(* IEC 61131-3 sources: plc_generation_empirical_study/datasets/task_bank_c06_formal_core_runtime_v0_4/tasks/C06_W25_lean_composite, 2 files *)

(* ---- interface.st ---- *)
FUNCTION_BLOCK C06_W25_lean_composite
VAR_INPUT
    A_Ch1 : BOOL;
    A_Ch2 : BOOL;
    A_Ch3 : BOOL;
    A_AutoMode : BOOL;
    A_AutoRequest : BOOL;
    A_ManualRequest : BOOL;
    A_BypassRequest : BOOL;
    A_BypassPermit : BOOL;
    A_SafetyOK : BOOL;
    A_Reset : BOOL;
    B_ItemPulse : BOOL;
    B_Rejected : BOOL;
    B_Stop : BOOL;
    B_Reset : BOOL;
    B_Target : INT;
    B_RejectLimit : INT;
    SubsystemBEnable : BOOL;
    CrossReset : BOOL;
END_VAR
VAR_OUTPUT
    A_RunPermit : BOOL;
    A_Degraded : BOOL;
    A_BypassActive : BOOL;
    A_Blocked : BOOL;
    B_AcceptedCount : INT;
    B_RejectCount : INT;
    B_ConsecutiveRejects : INT;
    B_Complete : BOOL;
    B_LockedOut : BOOL;
    CrossReady : BOOL;
    CrossBlocked : BOOL;
END_VAR
END_FUNCTION_BLOCK

(* ---- reference.st ---- *)
FUNCTION_BLOCK C06_W25_lean_composite
VAR_INPUT
    A_Ch1 : BOOL;
    A_Ch2 : BOOL;
    A_Ch3 : BOOL;
    A_AutoMode : BOOL;
    A_AutoRequest : BOOL;
    A_ManualRequest : BOOL;
    A_BypassRequest : BOOL;
    A_BypassPermit : BOOL;
    A_SafetyOK : BOOL;
    A_Reset : BOOL;
    B_ItemPulse : BOOL;
    B_Rejected : BOOL;
    B_Stop : BOOL;
    B_Reset : BOOL;
    B_Target : INT;
    B_RejectLimit : INT;
    SubsystemBEnable : BOOL;
    CrossReset : BOOL;
END_VAR
VAR_OUTPUT
    A_RunPermit : BOOL;
    A_Degraded : BOOL;
    A_BypassActive : BOOL;
    A_Blocked : BOOL;
    B_AcceptedCount : INT;
    B_RejectCount : INT;
    B_ConsecutiveRejects : INT;
    B_Complete : BOOL;
    B_LockedOut : BOOL;
    CrossReady : BOOL;
    CrossBlocked : BOOL;
END_VAR
VAR
    A_SelectedRequest : BOOL;
    A_VoteOK : BOOL;
    A_AnyChannel : BOOL;
    A_Unanimous : BOOL;
    B_PrevItem : BOOL;
END_VAR

A_SelectedRequest := (A_AutoMode AND A_AutoRequest) OR ((NOT A_AutoMode) AND A_ManualRequest);
A_VoteOK := (A_Ch1 AND A_Ch2) OR (A_Ch1 AND A_Ch3) OR (A_Ch2 AND A_Ch3);
A_AnyChannel := A_Ch1 OR A_Ch2 OR A_Ch3;
A_Unanimous := (A_Ch1 AND A_Ch2 AND A_Ch3) OR ((NOT A_Ch1) AND (NOT A_Ch2) AND (NOT A_Ch3));
IF A_Reset AND (NOT A_AutoRequest) AND (NOT A_ManualRequest) THEN
    A_BypassActive := FALSE;
ELSIF (NOT A_AutoMode) AND A_BypassRequest AND A_BypassPermit AND A_SafetyOK AND A_AnyChannel THEN
    A_BypassActive := TRUE;
END_IF;
A_RunPermit := A_SelectedRequest AND A_SafetyOK AND (A_VoteOK OR A_BypassActive);
A_Degraded := A_RunPermit AND ((NOT A_Unanimous) OR A_BypassActive);
A_Blocked := A_SelectedRequest AND (NOT A_RunPermit);

IF CrossReset THEN
    CrossReady := FALSE;
ELSIF A_RunPermit THEN
    CrossReady := TRUE;
END_IF;
CrossBlocked := SubsystemBEnable AND (NOT CrossReady);

IF SubsystemBEnable AND CrossReady THEN
    IF B_Reset AND B_Stop AND (NOT B_ItemPulse) THEN
        B_AcceptedCount := 0;
        B_RejectCount := 0;
        B_ConsecutiveRejects := 0;
        B_Complete := FALSE;
        B_LockedOut := FALSE;
    ELSIF B_RejectLimit <= 0 THEN
        B_LockedOut := TRUE;
    ELSIF B_ItemPulse AND (NOT B_PrevItem) AND (NOT B_Stop) AND (NOT B_Complete) AND (NOT B_LockedOut) THEN
        IF B_Rejected THEN
            B_RejectCount := B_RejectCount + 1;
            B_ConsecutiveRejects := B_ConsecutiveRejects + 1;
            IF B_ConsecutiveRejects >= B_RejectLimit THEN B_LockedOut := TRUE; END_IF;
        ELSE
            B_AcceptedCount := B_AcceptedCount + 1;
            B_ConsecutiveRejects := 0;
            IF (B_Target > 0) AND (B_AcceptedCount >= B_Target) THEN B_Complete := TRUE; END_IF;
        END_IF;
    END_IF;
    B_PrevItem := B_ItemPulse;
ELSE
    B_AcceptedCount := 0;
    B_RejectCount := 0;
    B_ConsecutiveRejects := 0;
    B_Complete := FALSE;
    B_LockedOut := FALSE;
END_IF;

END_FUNCTION_BLOCK
